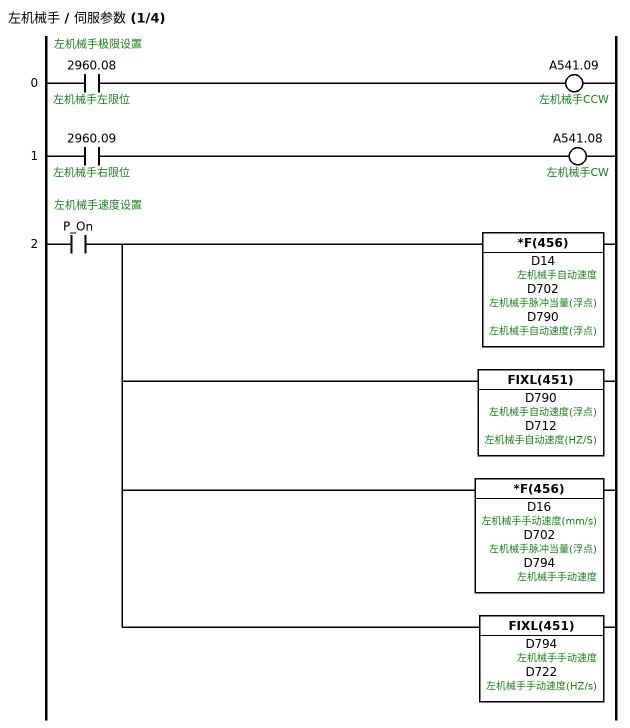
; [picture p137: 左机械手 / 伺服参数, rungs 0-2]
; rung 0: 左机械手极限设置
LD 2960.08  ; 左机械手左限位
OUT A541.09  ; 左机械手CCW
; rung 1
LD 2960.09  ; 左机械手右限位
OUT A541.08  ; 左机械手CW
; rung 2: 左机械手速度设置
LD P_On
*F(456) D14 D702 D790  ; 左机械手自动速度, 左机械手脉冲当量(浮点), 左机械手自动速度(浮点)
FIXL(451) D790 D712  ; 左机械手自动速度(浮点), 左机械手自动速度(HZ/S)
*F(456) D16 D702 D794  ; 左机械手手动速度(mm/s), 左机械手脉冲当量(浮点), 左机械手手动速度
FIXL(451) D794 D722  ; 左机械手手动速度, 左机械手手动速度(HZ/s)

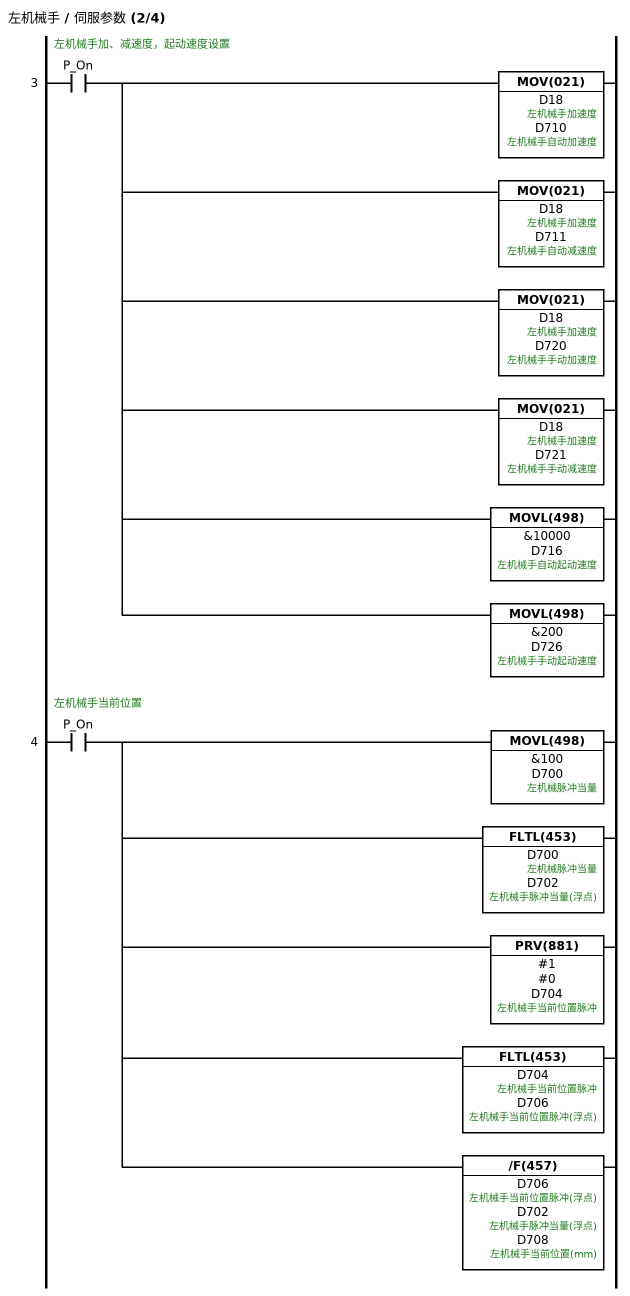
; rung 3: 左机械手加、减速度，起动速度设置
LD P_On
MOV(021) D18 D710  ; 左机械手加速度, 左机械手自动加速度
MOV(021) D18 D711  ; 左机械手加速度, 左机械手自动减速度
MOV(021) D18 D720  ; 左机械手加速度, 左机械手手动加速度
MOV(021) D18 D721  ; 左机械手加速度, 左机械手手动减速度
MOVL(498) &10000 D716  ; 左机械手自动起动速度
MOVL(498) &200 D726  ; 左机械手手动起动速度
; rung 4: 左机械手当前位置
LD P_On
MOVL(498) &100 D700  ; 左机械脉冲当量
FLTL(453) D700 D702  ; 左机械脉冲当量, 左机械手脉冲当量(浮点)
PRV(881) #1 #0 D704  ; 左机械手当前位置脉冲
FLTL(453) D704 D706  ; 左机械手当前位置脉冲, 左机械手当前位置脉冲(浮点)
/F(457) D706 D702 D708  ; 左机械手当前位置脉冲(浮点), 左机械手脉冲当量(浮点), 左机械手当前位置(mm)

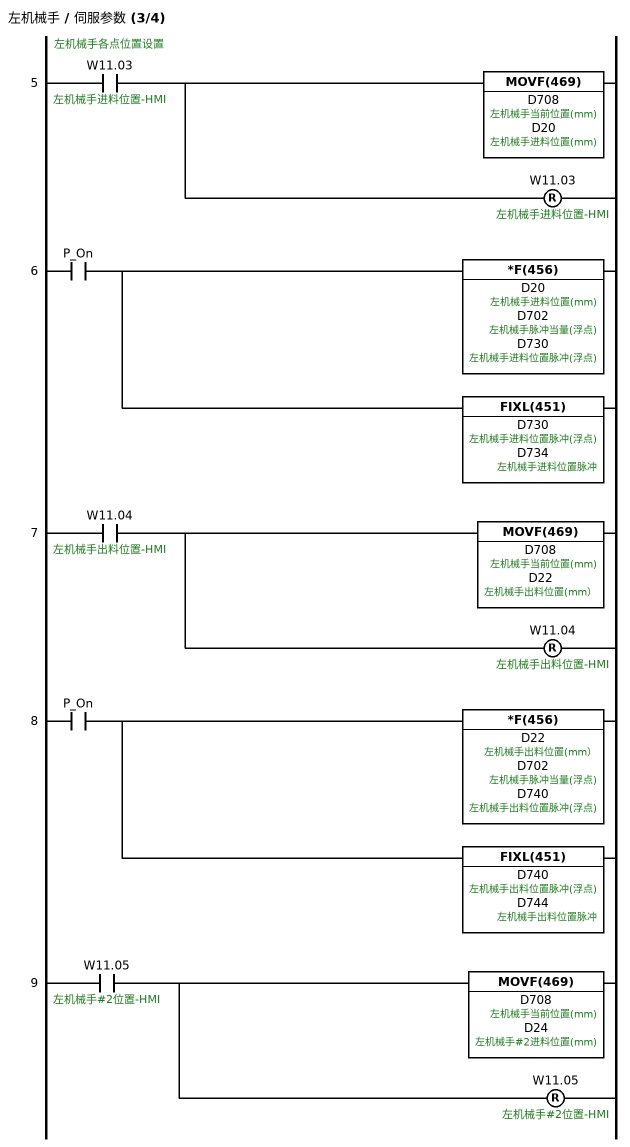
; rung 5: 左机械手各点位置设置
LD W11.03  ; 左机械手进料位置-HMI
MOVF(469) D708 D20  ; 左机械手当前位置(mm), 左机械手进料位置(mm)
RSET W11.03  ; 左机械手进料位置-HMI
; rung 6
LD P_On
*F(456) D20 D702 D730  ; 左机械手进料位置(mm), 左机械手脉冲当量(浮点), 左机械手进料位置脉冲(浮点)
FIXL(451) D730 D734  ; 左机械手进料位置脉冲(浮点), 左机械手进料位置脉冲
; rung 7
LD W11.04  ; 左机械手出料位置-HMI
MOVF(469) D708 D22  ; 左机械手当前位置(mm), 左机械手出料位置(mm）
RSET W11.04  ; 左机械手出料位置-HMI
; rung 8
LD P_On
*F(456) D22 D702 D740  ; 左机械手出料位置(mm）, 左机械手脉冲当量(浮点), 左机械手出料位置脉冲(浮点)
FIXL(451) D740 D744  ; 左机械手出料位置脉冲(浮点), 左机械手出料位置脉冲
; rung 9
LD W11.05  ; 左机械手#2位置-HMI
MOVF(469) D708 D24  ; 左机械手当前位置(mm), 左机械手#2进料位置(mm)
RSET W11.05  ; 左机械手#2位置-HMI

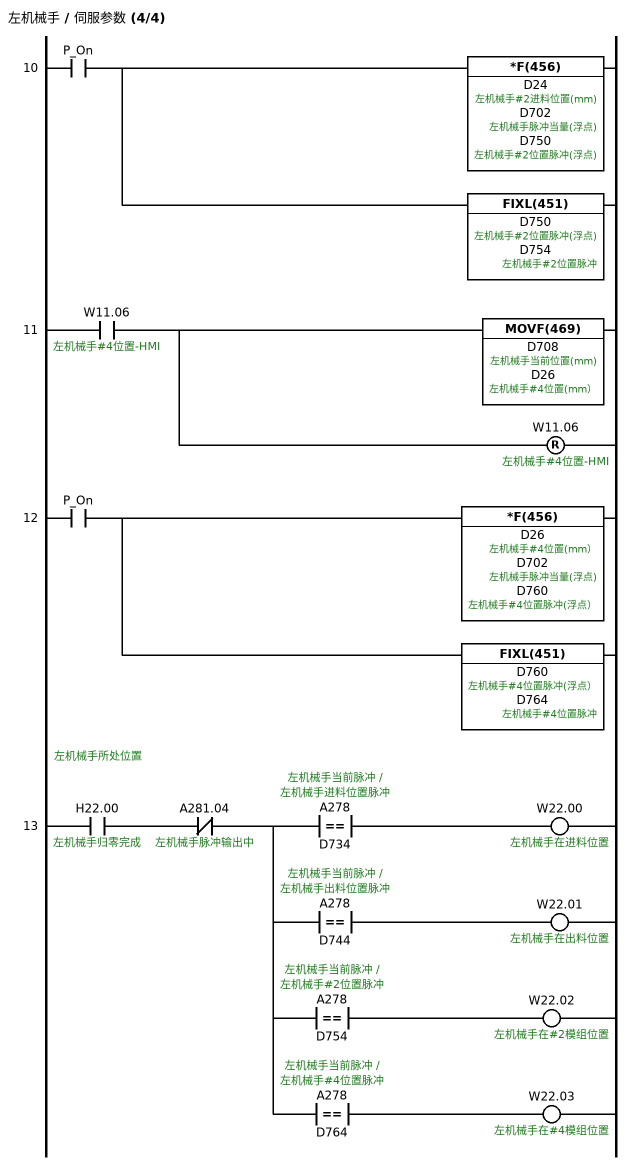
; rung 10
LD P_On
*F(456) D24 D702 D750  ; 左机械手#2进料位置(mm), 左机械手脉冲当量(浮点), 左机械手#2位置脉冲(浮点)
FIXL(451) D750 D754  ; 左机械手#2位置脉冲(浮点), 左机械手#2位置脉冲
; rung 11
LD W11.06  ; 左机械手#4位置-HMI
MOVF(469) D708 D26  ; 左机械手当前位置(mm), 左机械手#4位置(mm）
RSET W11.06  ; 左机械手#4位置-HMI
; rung 12
LD P_On
*F(456) D26 D702 D760  ; 左机械手#4位置(mm）, 左机械手脉冲当量(浮点), 左机械手#4位置脉冲(浮点）
FIXL(451) D760 D764  ; 左机械手#4位置脉冲(浮点）, 左机械手#4位置脉冲
; rung 13: 左机械手所处位置
LD H22.00  ; 左机械手归零完成
ANDNOT A281.04  ; 左机械手脉冲输出中
OUT TR0
AND=SL(303) A278 D734  ; 左机械手当前脉冲, 左机械手进料位置脉冲
OUT W22.00  ; 左机械手在进料位置
LD TR0
AND=SL(303) A278 D744  ; 左机械手当前脉冲, 左机械手出料位置脉冲
OUT W22.01  ; 左机械手在出料位置
LD TR0
AND=SL(303) A278 D754  ; 左机械手当前脉冲, 左机械手#2位置脉冲
OUT W22.02  ; 左机械手在#2模组位置
LD TR0
AND=SL(303) A278 D764  ; 左机械手当前脉冲, 左机械手#4位置脉冲
OUT W22.03  ; 左机械手在#4模组位置

### Section 轴控运动及外部输出

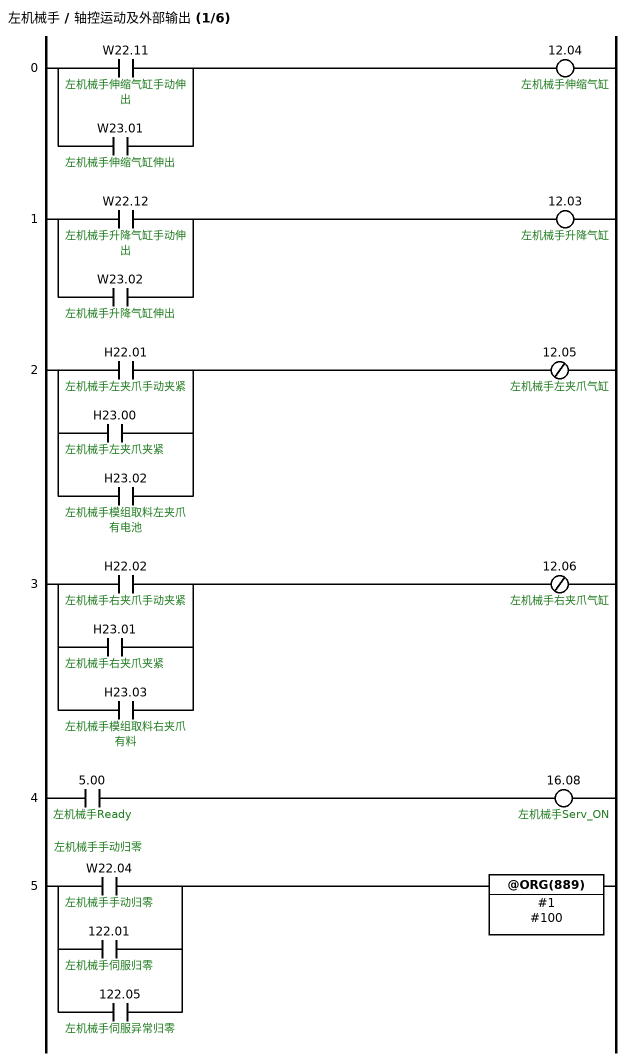
; rung 0
LD W22.11  ; 左机械手伸缩气缸手动伸出
OR W23.01  ; 左机械手伸缩气缸伸出
OUT 12.04  ; 左机械手伸缩气缸
; rung 1
LD W22.12  ; 左机械手升降气缸手动伸出
OR W23.02  ; 左机械手升降气缸伸出
OUT 12.03  ; 左机械手升降气缸
; rung 2
LD H22.01  ; 左机械手左夹爪手动夹紧
OR H23.00  ; 左机械手左夹爪夹紧
OR H23.02  ; 左机械手模组取料左夹爪有电池
OUTNOT 12.05  ; 左机械手左夹爪气缸
; rung 3
LD H22.02  ; 左机械手右夹爪手动夹紧
OR H23.01  ; 左机械手右夹爪夹紧
OR H23.03  ; 左机械手模组取料右夹爪有料
OUTNOT 12.06  ; 左机械手右夹爪气缸
; rung 4
LD 5.00  ; 左机械手Ready
OUT 16.08  ; 左机械手Serv_ON
; rung 5: 左机械手手动归零
LD W22.04  ; 左机械手手动归零
OR 122.01  ; 左机械手伺服归零
OR 122.05  ; 左机械手伺服异常归零
@ORG(889) #1 #100

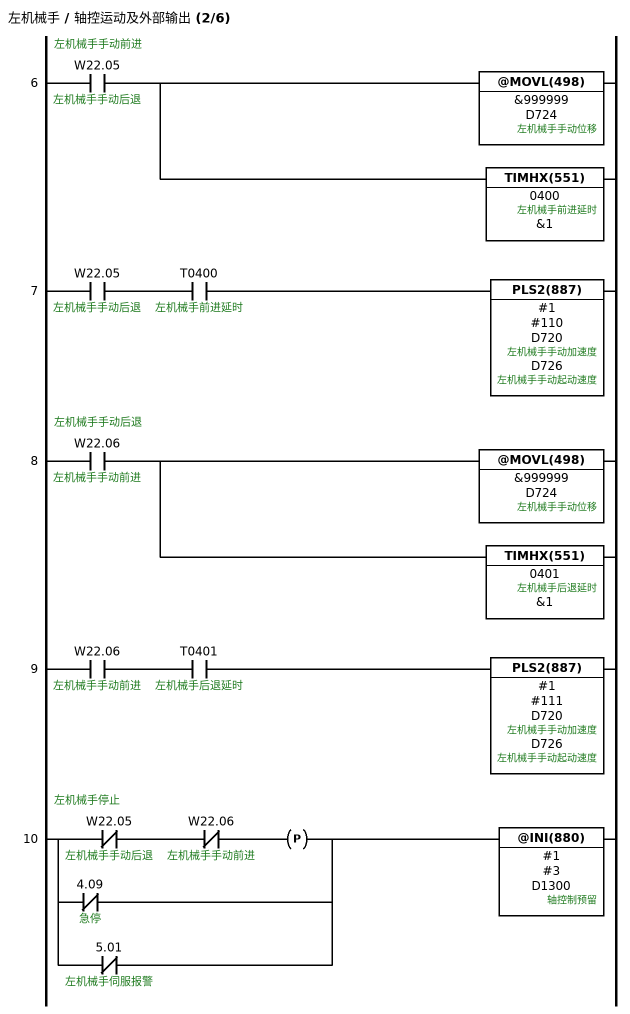
; rung 6: 左机械手手动前进
LD W22.05  ; 左机械手手动后退
@MOVL(498) &999999 D724  ; 左机械手手动位移
TIMHX(551) 0400 &1  ; 左机械手前进延时
; rung 7
LD W22.05  ; 左机械手手动后退
AND T0400  ; 左机械手前进延时
PLS2(887) #1 #110 D720 D726  ; 左机械手手动加速度, 左机械手手动起动速度
; rung 8: 左机械手手动后退
LD W22.06  ; 左机械手手动前进
@MOVL(498) &999999 D724  ; 左机械手手动位移
TIMHX(551) 0401 &1  ; 左机械手后退延时
; rung 9
LD W22.06  ; 左机械手手动前进
AND T0401  ; 左机械手后退延时
PLS2(887) #1 #111 D720 D726  ; 左机械手手动加速度, 左机械手手动起动速度
; rung 10: 左机械手停止
LDNOT W22.05  ; 左机械手手动后退
ANDNOT W22.06  ; 左机械手手动前进
UP(521)
ORNOT 4.09  ; 急停
ORNOT 5.01  ; 左机械手伺服报警
@INI(880) #1 #3 D1300  ; 轴控制预留

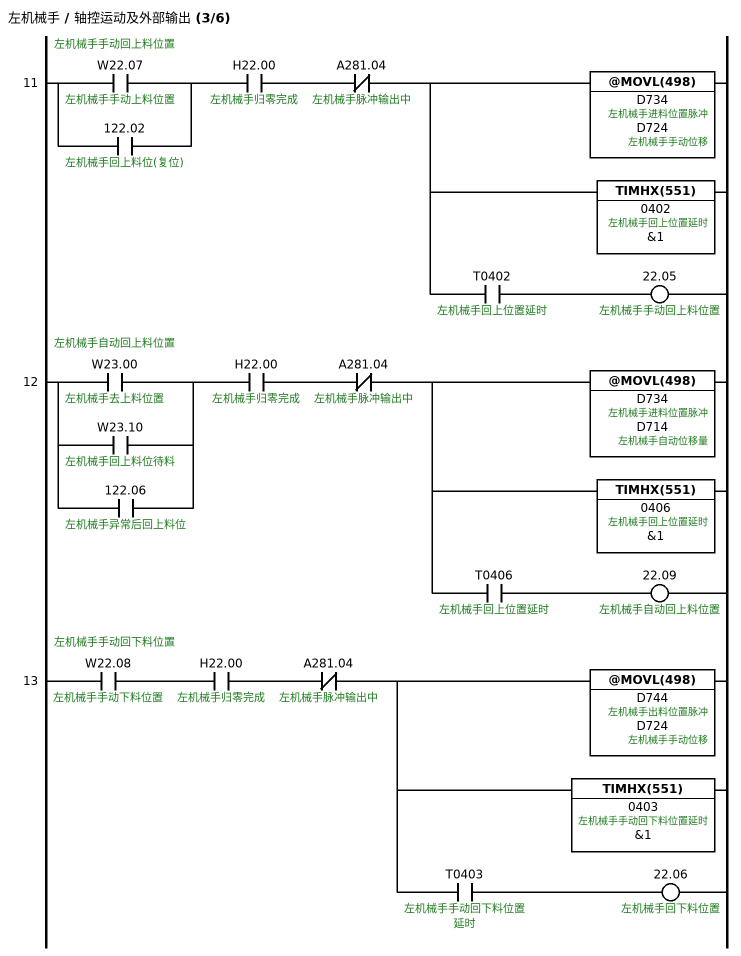
; rung 11: 左机械手手动回上料位置
LD W22.07  ; 左机械手手动上料位置
OR 122.02  ; 左机械手回上料位(复位)
AND H22.00  ; 左机械手归零完成
ANDNOT A281.04  ; 左机械手脉冲输出中
@MOVL(498) D734 D724  ; 左机械手进料位置脉冲, 左机械手手动位移
TIMHX(551) 0402 &1  ; 左机械手回上位置延时
AND T0402  ; 左机械手回上位置延时
OUT 22.05  ; 左机械手手动回上料位置
; rung 12: 左机械手自动回上料位置
LD W23.00  ; 左机械手去上料位置
OR W23.10  ; 左机械手回上料位待料
OR 122.06  ; 左机械手异常后回上料位
AND H22.00  ; 左机械手归零完成
ANDNOT A281.04  ; 左机械手脉冲输出中
@MOVL(498) D734 D714  ; 左机械手进料位置脉冲, 左机械手自动位移量
TIMHX(551) 0406 &1  ; 左机械手回上位置延时
AND T0406  ; 左机械手回上位置延时
OUT 22.09  ; 左机械手自动回上料位置
; rung 13: 左机械手手动回下料位置
LD W22.08  ; 左机械手手动下料位置
AND H22.00  ; 左机械手归零完成
ANDNOT A281.04  ; 左机械手脉冲输出中
@MOVL(498) D744 D724  ; 左机械手出料位置脉冲, 左机械手手动位移
TIMHX(551) 0403 &1  ; 左机械手手动回下料位置延时
AND T0403  ; 左机械手手动回下料位置延时
OUT 22.06  ; 左机械手回下料位置

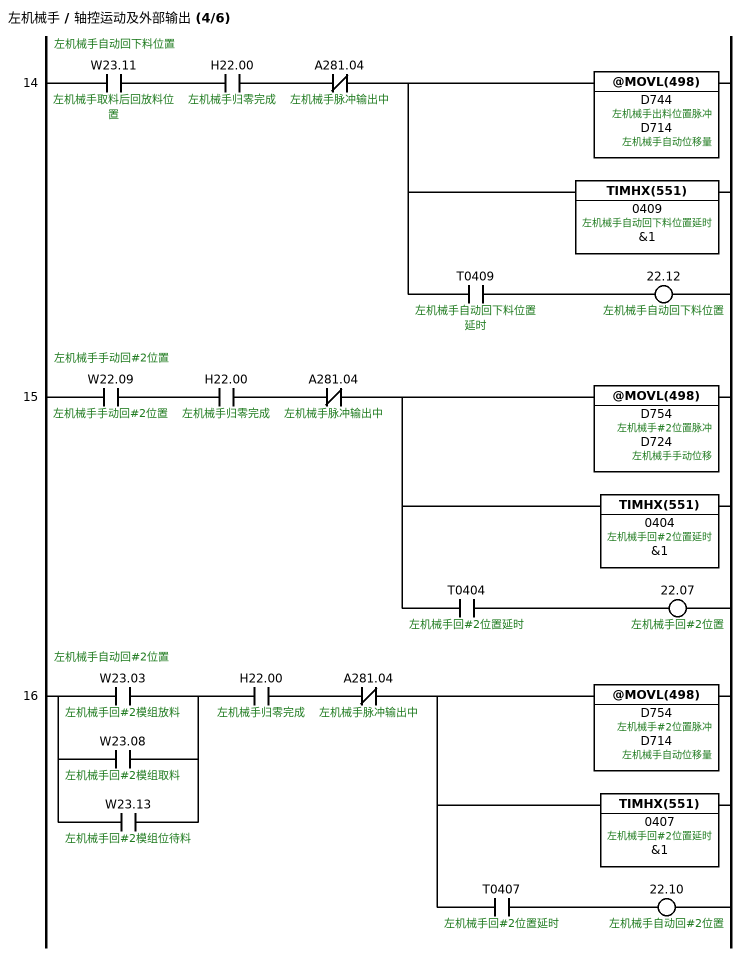
; rung 14: 左机械手自动回下料位置
LD W23.11  ; 左机械手取料后回放料位置
AND H22.00  ; 左机械手归零完成
ANDNOT A281.04  ; 左机械手脉冲输出中
@MOVL(498) D744 D714  ; 左机械手出料位置脉冲, 左机械手自动位移量
TIMHX(551) 0409 &1  ; 左机械手自动回下料位置延时
AND T0409  ; 左机械手自动回下料位置延时
OUT 22.12  ; 左机械手自动回下料位置
; rung 15: 左机械手手动回#2位置
LD W22.09  ; 左机械手手动回#2位置
AND H22.00  ; 左机械手归零完成
ANDNOT A281.04  ; 左机械手脉冲输出中
@MOVL(498) D754 D724  ; 左机械手#2位置脉冲, 左机械手手动位移
TIMHX(551) 0404 &1  ; 左机械手回#2位置延时
AND T0404  ; 左机械手回#2位置延时
OUT 22.07  ; 左机械手回#2位置
; rung 16: 左机械手自动回#2位置
LD W23.03  ; 左机械手回#2模组放料
OR W23.08  ; 左机械手回#2模组取料
OR W23.13  ; 左机械手回#2模组位待料
AND H22.00  ; 左机械手归零完成
ANDNOT A281.04  ; 左机械手脉冲输出中
@MOVL(498) D754 D714  ; 左机械手#2位置脉冲, 左机械手自动位移量
TIMHX(551) 0407 &1  ; 左机械手回#2位置延时
AND T0407  ; 左机械手回#2位置延时
OUT 22.10  ; 左机械手自动回#2位置

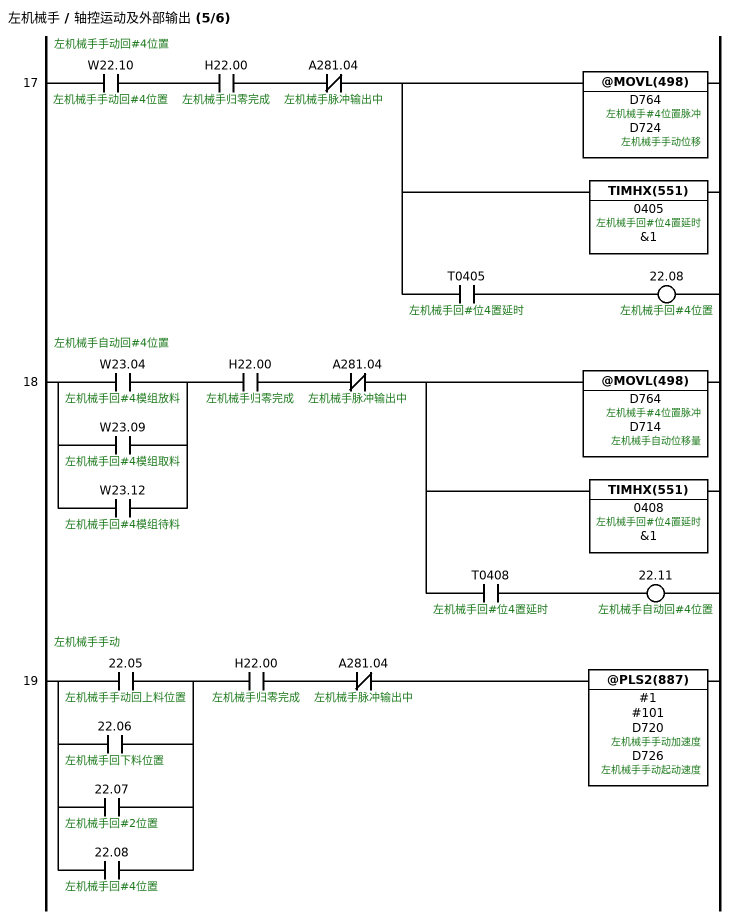
; rung 17: 左机械手手动回#4位置
LD W22.10  ; 左机械手手动回#4位置
AND H22.00  ; 左机械手归零完成
ANDNOT A281.04  ; 左机械手脉冲输出中
@MOVL(498) D764 D724  ; 左机械手#4位置脉冲, 左机械手手动位移
TIMHX(551) 0405 &1  ; 左机械手回#位4置延时
AND T0405  ; 左机械手回#位4置延时
OUT 22.08  ; 左机械手回#4位置
; rung 18: 左机械手自动回#4位置
LD W23.04  ; 左机械手回#4模组放料
OR W23.09  ; 左机械手回#4模组取料
OR W23.12  ; 左机械手回#4模组待料
AND H22.00  ; 左机械手归零完成
ANDNOT A281.04  ; 左机械手脉冲输出中
@MOVL(498) D764 D714  ; 左机械手#4位置脉冲, 左机械手自动位移量
TIMHX(551) 0408 &1  ; 左机械手回#位4置延时
AND T0408  ; 左机械手回#位4置延时
OUT 22.11  ; 左机械手自动回#4位置
; rung 19: 左机械手手动
LD 22.05  ; 左机械手手动回上料位置
OR 22.06  ; 左机械手回下料位置
OR 22.07  ; 左机械手回#2位置
OR 22.08  ; 左机械手回#4位置
AND H22.00  ; 左机械手归零完成
ANDNOT A281.04  ; 左机械手脉冲输出中
@PLS2(887) #1 #101 D720 D726  ; 左机械手手动加速度, 左机械手手动起动速度

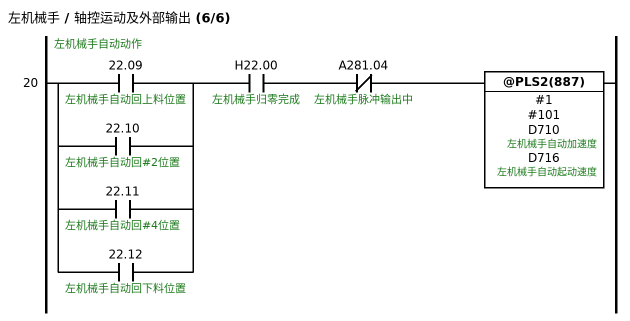
; rung 20: 左机械手自动动作
LD 22.09  ; 左机械手自动回上料位置
OR 22.10  ; 左机械手自动回#2位置
OR 22.11  ; 左机械手自动回#4位置
OR 22.12  ; 左机械手自动回下料位置
AND H22.00  ; 左机械手归零完成
ANDNOT A281.04  ; 左机械手脉冲输出中
@PLS2(887) #1 #101 D710 D716  ; 左机械手自动加速度, 左机械手自动起动速度

### Section 自动报警

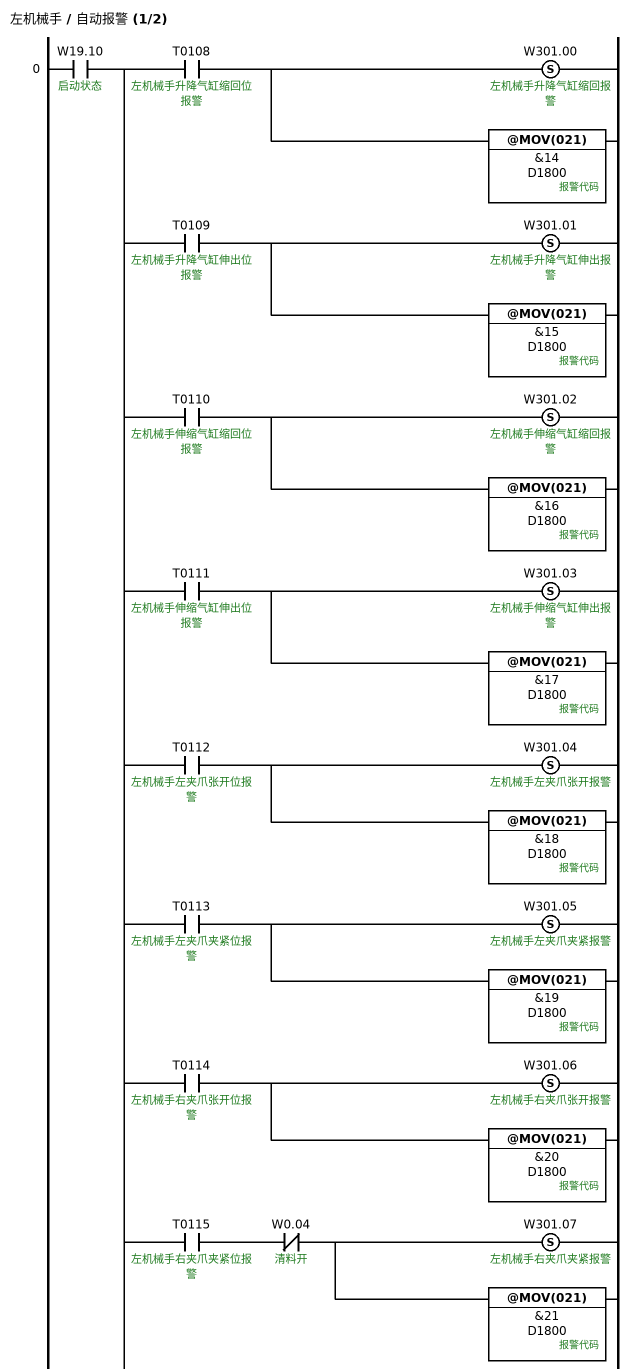

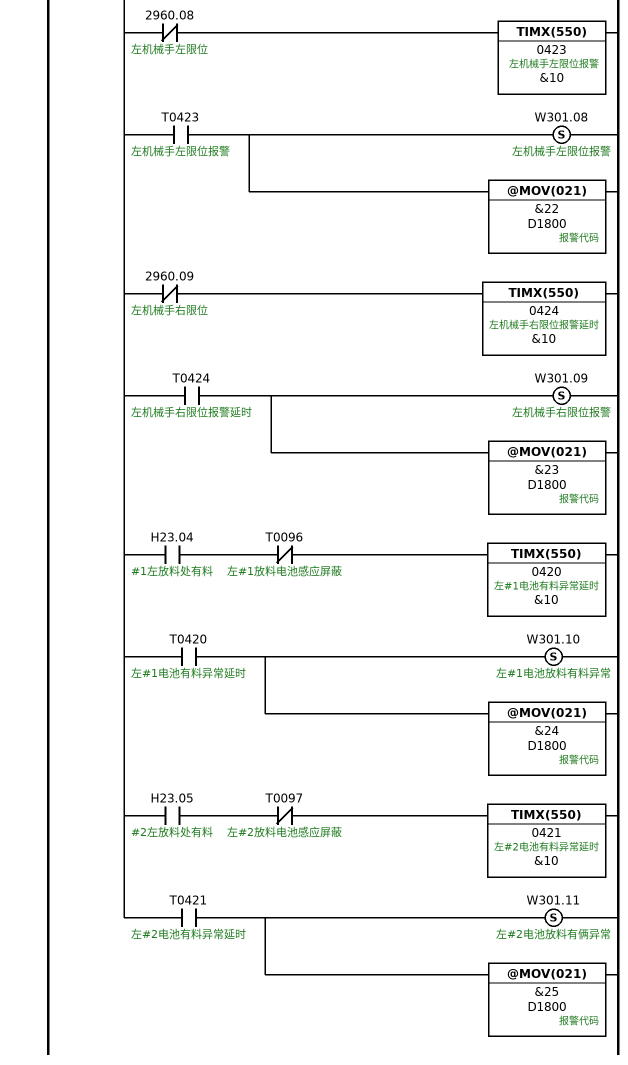
; rung 0
LD W19.10  ; 启动状态
OUT TR0
AND T0108  ; 左机械手升降气缸缩回位报警
SET W301.00  ; 左机械手升降气缸缩回报警
@MOV(021) &14 D1800  ; 报警代码
LD TR0
AND T0109  ; 左机械手升降气缸伸出位报警
SET W301.01  ; 左机械手升降气缸伸出报警
@MOV(021) &15 D1800  ; 报警代码
LD TR0
AND T0110  ; 左机械手伸缩气缸缩回位报警
SET W301.02  ; 左机械手伸缩气缸缩回报警
@MOV(021) &16 D1800  ; 报警代码
LD TR0
AND T0111  ; 左机械手伸缩气缸伸出位报警
SET W301.03  ; 左机械手伸缩气缸伸出报警
@MOV(021) &17 D1800  ; 报警代码
LD TR0
AND T0112  ; 左机械手左夹爪张开位报警
SET W301.04  ; 左机械手左夹爪张开报警
@MOV(021) &18 D1800  ; 报警代码
LD TR0
AND T0113  ; 左机械手左夹爪夹紧位报警
SET W301.05  ; 左机械手左夹爪夹紧报警
@MOV(021) &19 D1800  ; 报警代码
LD TR0
AND T0114  ; 左机械手右夹爪张开位报警
SET W301.06  ; 左机械手右夹爪张开报警
@MOV(021) &20 D1800  ; 报警代码
LD TR0
AND T0115  ; 左机械手右夹爪夹紧位报警
ANDNOT W0.04  ; 清料开
SET W301.07  ; 左机械手右夹爪夹紧报警
@MOV(021) &21 D1800  ; 报警代码
LD TR0
ANDNOT 2960.08  ; 左机械手左限位
TIMX(550) 0423 &10  ; 左机械手左限位报警
LD TR0
AND T0423  ; 左机械手左限位报警
SET W301.08  ; 左机械手左限位报警
@MOV(021) &22 D1800  ; 报警代码
LD TR0
ANDNOT 2960.09  ; 左机械手右限位
TIMX(550) 0424 &10  ; 左机械手右限位报警延时
LD TR0
AND T0424  ; 左机械手右限位报警延时
SET W301.09  ; 左机械手右限位报警
@MOV(021) &23 D1800  ; 报警代码
LD TR0
AND H23.04  ; #1左放料处有料
ANDNOT T0096  ; 左#1放料电池感应屏蔽
TIMX(550) 0420 &10  ; 左#1电池有料异常延时
LD TR0
AND T0420  ; 左#1电池有料异常延时
SET W301.10  ; 左#1电池放料有料异常
@MOV(021) &24 D1800  ; 报警代码
LD TR0
AND H23.05  ; #2左放料处有料
ANDNOT T0097  ; 左#2放料电池感应屏蔽
TIMX(550) 0421 &10  ; 左#2电池有料异常延时
LD TR0
AND T0421  ; 左#2电池有料异常延时
SET W301.11  ; 左#2电池放料有俩异常
@MOV(021) &25 D1800  ; 报警代码

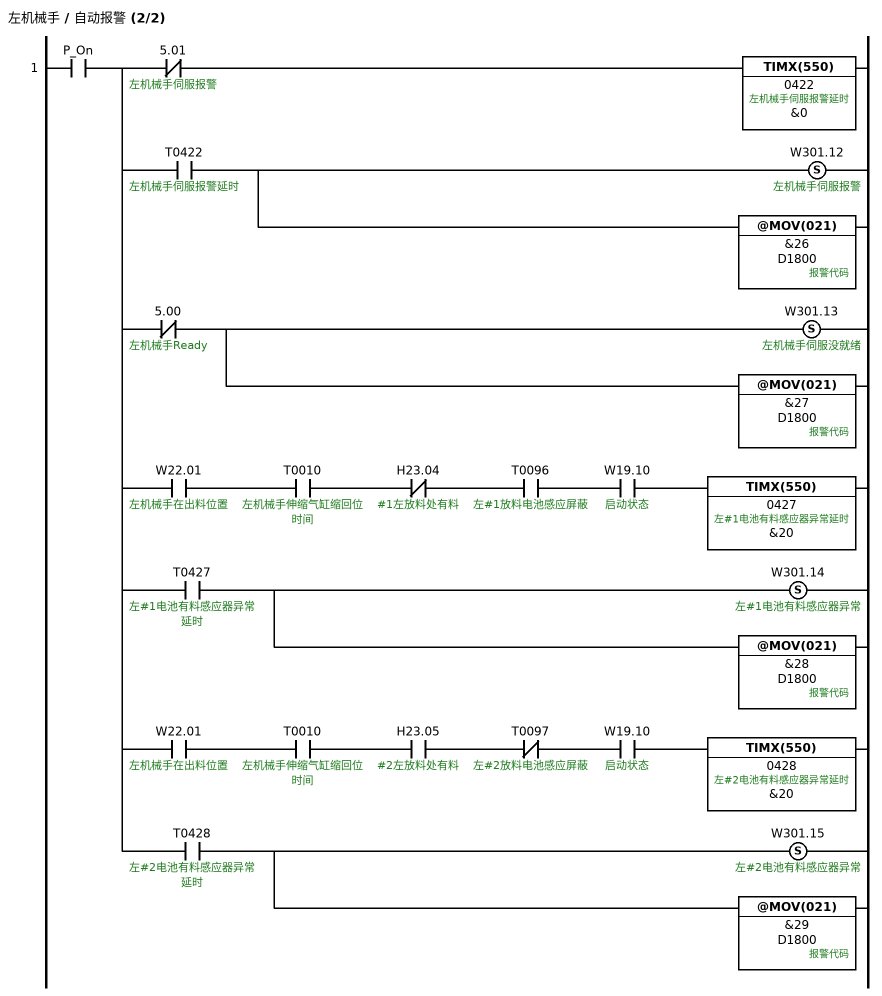
; rung 1
LD P_On
OUT TR0
ANDNOT 5.01  ; 左机械手伺服报警
TIMX(550) 0422 &0  ; 左机械手伺服报警延时
LD TR0
AND T0422  ; 左机械手伺服报警延时
SET W301.12  ; 左机械手伺服报警
@MOV(021) &26 D1800  ; 报警代码
LD TR0
ANDNOT 5.00  ; 左机械手Ready
SET W301.13  ; 左机械手伺服没就绪
@MOV(021) &27 D1800  ; 报警代码
LD TR0
AND W22.01  ; 左机械手在出料位置
AND T0010  ; 左机械手伸缩气缸缩回位时间
ANDNOT H23.04  ; #1左放料处有料
AND T0096  ; 左#1放料电池感应屏蔽
AND W19.10  ; 启动状态
TIMX(550) 0427 &20  ; 左#1电池有料感应器异常延时
LD TR0
AND T0427  ; 左#1电池有料感应器异常延时
SET W301.14  ; 左#1电池有料感应器异常
@MOV(021) &28 D1800  ; 报警代码
LD TR0
AND W22.01  ; 左机械手在出料位置
AND T0010  ; 左机械手伸缩气缸缩回位时间
AND H23.05  ; #2左放料处有料
ANDNOT T0097  ; 左#2放料电池感应屏蔽
AND W19.10  ; 启动状态
TIMX(550) 0428 &20  ; 左#2电池有料感应器异常延时
LD TR0
AND T0428  ; 左#2电池有料感应器异常延时
SET W301.15  ; 左#2电池有料感应器异常
@MOV(021) &29 D1800  ; 报警代码

### Section 左机械手复位

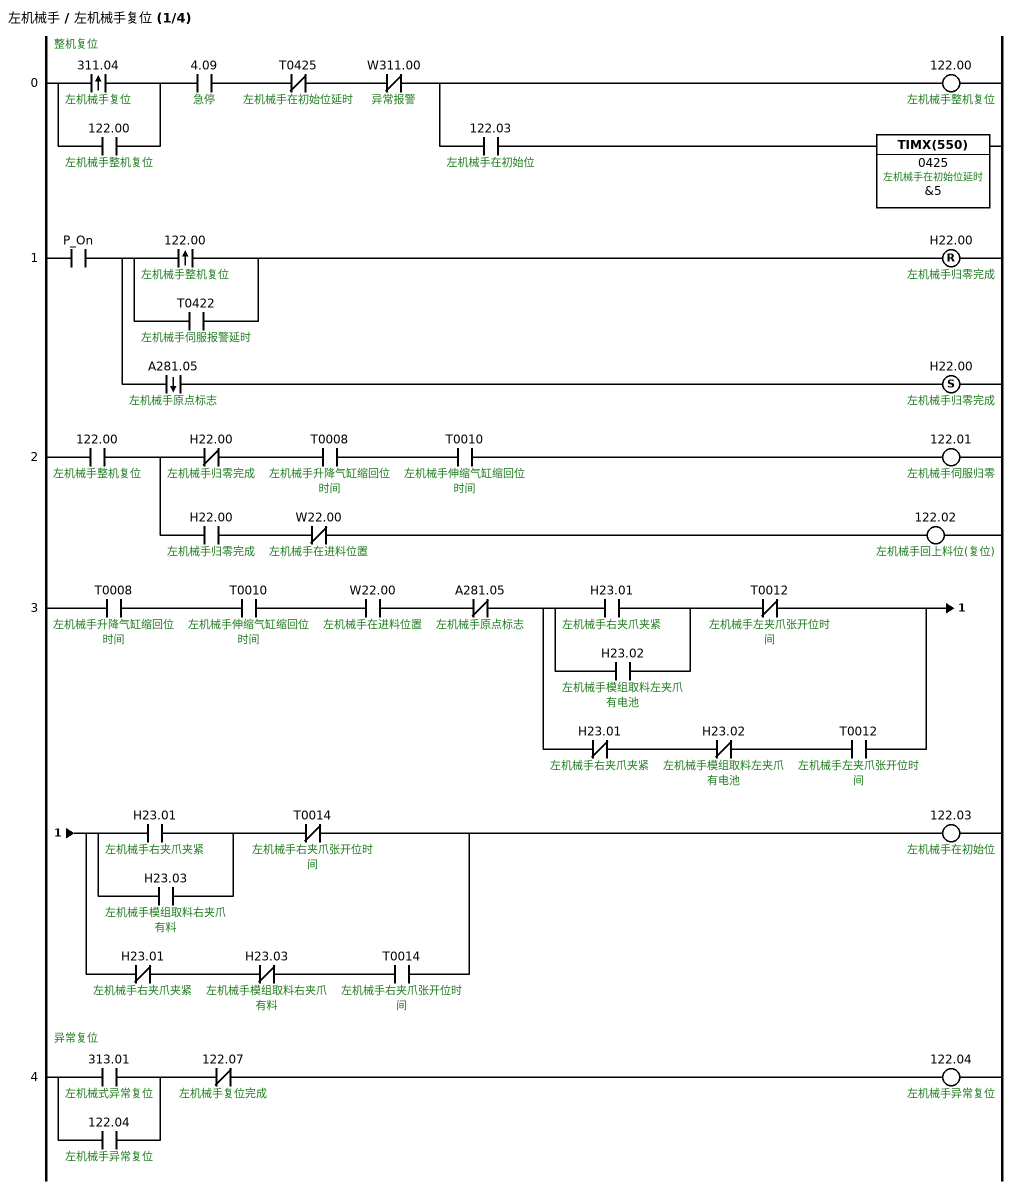
; rung 0: 整机复位
@LD 311.04  ; 左机械手复位
OR 122.00  ; 左机械手整机复位
AND 4.09  ; 急停
ANDNOT T0425  ; 左机械手在初始位延时
ANDNOT W311.00  ; 异常报警
OUT 122.00  ; 左机械手整机复位
AND 122.03  ; 左机械手在初始位
TIMX(550) 0425 &5  ; 左机械手在初始位延时
; rung 1
LD P_On
OUT TR0
@LD 122.00  ; 左机械手整机复位
OR T0422  ; 左机械手伺服报警延时
ANDLD
RSET H22.00  ; 左机械手归零完成
LD TR0
%AND A281.05  ; 左机械手原点标志
SET H22.00  ; 左机械手归零完成
; rung 2
LD 122.00  ; 左机械手整机复位
OUT TR0
ANDNOT H22.00  ; 左机械手归零完成
AND T0008  ; 左机械手升降气缸缩回位时间
AND T0010  ; 左机械手伸缩气缸缩回位时间
OUT 122.01  ; 左机械手伺服归零
LD TR0
AND H22.00  ; 左机械手归零完成
ANDNOT W22.00  ; 左机械手在进料位置
OUT 122.02  ; 左机械手回上料位(复位)
; rung 3
LD T0008  ; 左机械手升降气缸缩回位时间
AND T0010  ; 左机械手伸缩气缸缩回位时间
AND W22.00  ; 左机械手在进料位置
ANDNOT A281.05  ; 左机械手原点标志
LD H23.01  ; 左机械手右夹爪夹紧
OR H23.02  ; 左机械手模组取料左夹爪有电池
ANDNOT T0012  ; 左机械手左夹爪张开位时间
LDNOT H23.01  ; 左机械手右夹爪夹紧
ANDNOT H23.02  ; 左机械手模组取料左夹爪有电池
AND T0012  ; 左机械手左夹爪张开位时间
ORLD
ANDLD
LD H23.01  ; 左机械手右夹爪夹紧
OR H23.03  ; 左机械手模组取料右夹爪有料
ANDNOT T0014  ; 左机械手右夹爪张开位时间
LDNOT H23.01  ; 左机械手右夹爪夹紧
ANDNOT H23.03  ; 左机械手模组取料右夹爪有料
AND T0014  ; 左机械手右夹爪张开位时间
ORLD
ANDLD
OUT 122.03  ; 左机械手在初始位
; rung 4: 异常复位
LD 313.01  ; 左机械式异常复位
OR 122.04  ; 左机械手异常复位
ANDNOT 122.07  ; 左机械手复位完成
OUT 122.04  ; 左机械手异常复位

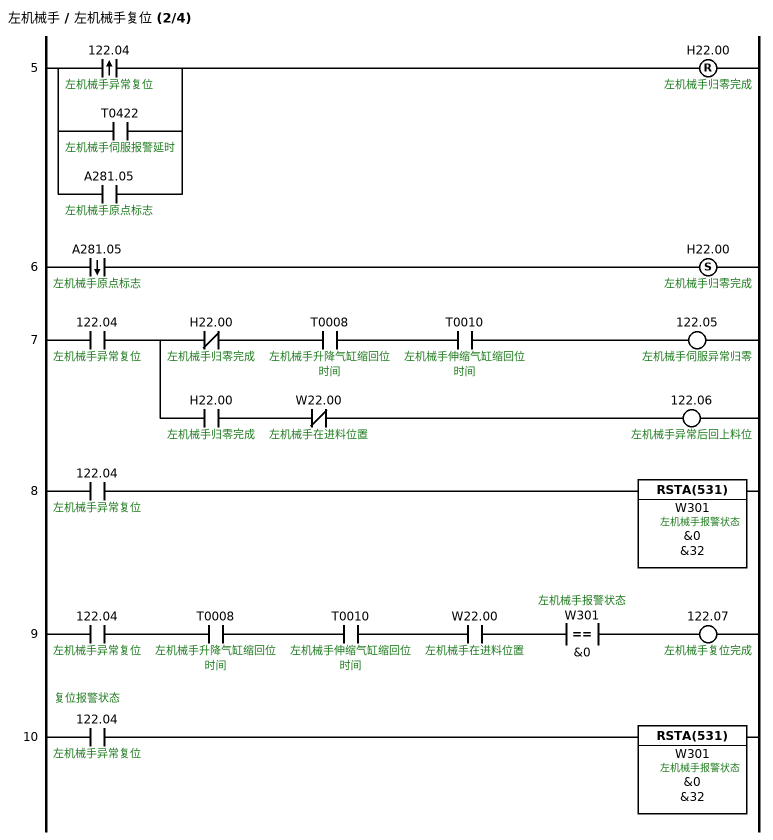
; rung 5
@LD 122.04  ; 左机械手异常复位
OR T0422  ; 左机械手伺服报警延时
OR A281.05  ; 左机械手原点标志
RSET H22.00  ; 左机械手归零完成
; rung 6
%LD A281.05  ; 左机械手原点标志
SET H22.00  ; 左机械手归零完成
; rung 7
LD 122.04  ; 左机械手异常复位
OUT TR0
ANDNOT H22.00  ; 左机械手归零完成
AND T0008  ; 左机械手升降气缸缩回位时间
AND T0010  ; 左机械手伸缩气缸缩回位时间
OUT 122.05  ; 左机械手伺服异常归零
LD TR0
AND H22.00  ; 左机械手归零完成
ANDNOT W22.00  ; 左机械手在进料位置
OUT 122.06  ; 左机械手异常后回上料位
; rung 8
LD 122.04  ; 左机械手异常复位
RSTA(531) W301 &0 &32  ; 左机械手报警状态
; rung 9
LD 122.04  ; 左机械手异常复位
AND T0008  ; 左机械手升降气缸缩回位时间
AND T0010  ; 左机械手伸缩气缸缩回位时间
AND W22.00  ; 左机械手在进料位置
AND=L(301) W301 &0  ; 左机械手报警状态
OUT 122.07  ; 左机械手复位完成
; rung 10: 复位报警状态
LD 122.04  ; 左机械手异常复位
RSTA(531) W301 &0 &32  ; 左机械手报警状态

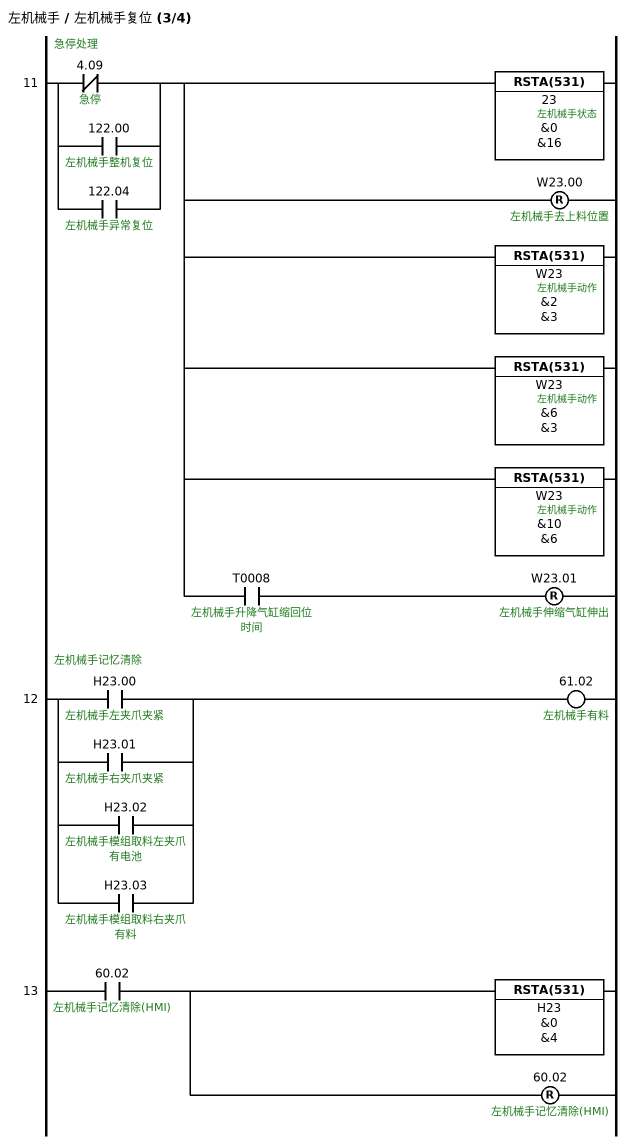
; rung 11: 急停处理
LDNOT 4.09  ; 急停
OR 122.00  ; 左机械手整机复位
OR 122.04  ; 左机械手异常复位
RSTA(531) 23 &0 &16  ; 左机械手状态
RSET W23.00  ; 左机械手去上料位置
RSTA(531) W23 &2 &3  ; 左机械手动作
RSTA(531) W23 &6 &3  ; 左机械手动作
RSTA(531) W23 &10 &6  ; 左机械手动作
AND T0008  ; 左机械手升降气缸缩回位时间
RSET W23.01  ; 左机械手伸缩气缸伸出
; rung 12: 左机械手记忆清除
LD H23.00  ; 左机械手左夹爪夹紧
OR H23.01  ; 左机械手右夹爪夹紧
OR H23.02  ; 左机械手模组取料左夹爪有电池
OR H23.03  ; 左机械手模组取料右夹爪有料
OUT 61.02  ; 左机械手有料
; rung 13
LD 60.02  ; 左机械手记忆清除(HMI)
RSTA(531) H23 &0 &4
RSET 60.02  ; 左机械手记忆清除(HMI)

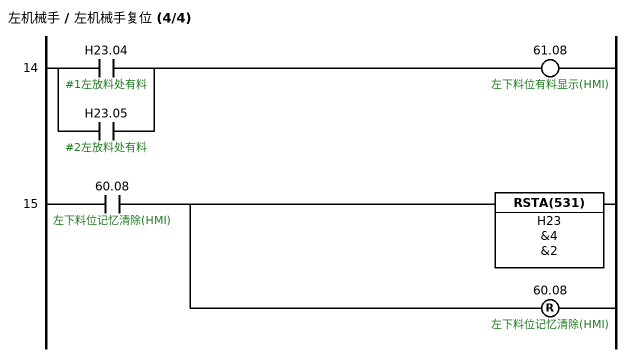
; rung 14
LD H23.04  ; #1左放料处有料
OR H23.05  ; #2左放料处有料
OUT 61.08  ; 左下料位有料显示(HMI)
; rung 15
LD 60.08  ; 左下料位记忆清除(HMI)
RSTA(531) H23 &4 &2
RSET 60.08  ; 左下料位记忆清除(HMI)

### Section END
; rung 0
END(001)

## Program 右机械手 (cyclic task 5)

### Section 右机械手手动

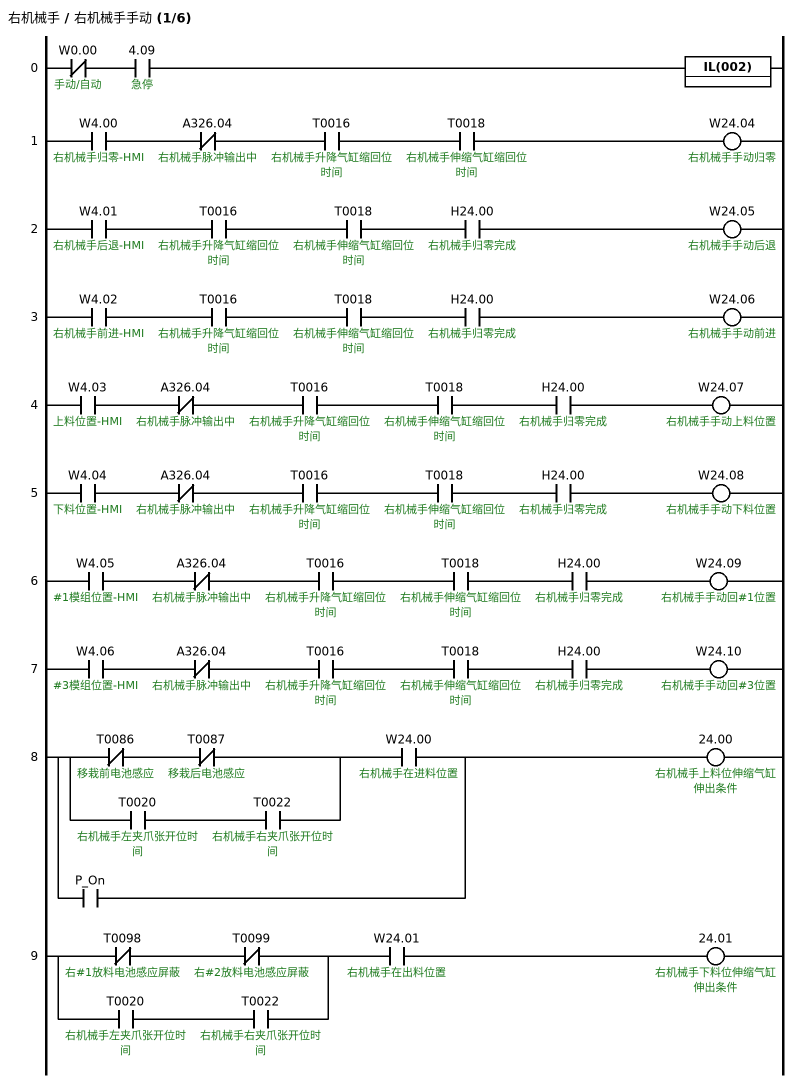
; rung 0
LDNOT W0.00  ; 手动/自动
AND 4.09  ; 急停
IL(002)
; rung 1
LD W4.00  ; 右机械手归零-HMI
ANDNOT A326.04  ; 右机械手脉冲输出中
AND T0016  ; 右机械手升降气缸缩回位时间
AND T0018  ; 右机械手伸缩气缸缩回位时间
OUT W24.04  ; 右机械手手动归零
; rung 2
LD W4.01  ; 右机械手后退-HMI
AND T0016  ; 右机械手升降气缸缩回位时间
AND T0018  ; 右机械手伸缩气缸缩回位时间
AND H24.00  ; 右机械手归零完成
OUT W24.05  ; 右机械手手动后退
; rung 3
LD W4.02  ; 右机械手前进-HMI
AND T0016  ; 右机械手升降气缸缩回位时间
AND T0018  ; 右机械手伸缩气缸缩回位时间
AND H24.00  ; 右机械手归零完成
OUT W24.06  ; 右机械手手动前进
; rung 4
LD W4.03  ; 上料位置-HMI
ANDNOT A326.04  ; 右机械手脉冲输出中
AND T0016  ; 右机械手升降气缸缩回位时间
AND T0018  ; 右机械手伸缩气缸缩回位时间
AND H24.00  ; 右机械手归零完成
OUT W24.07  ; 右机械手手动上料位置
; rung 5
LD W4.04  ; 下料位置-HMI
ANDNOT A326.04  ; 右机械手脉冲输出中
AND T0016  ; 右机械手升降气缸缩回位时间
AND T0018  ; 右机械手伸缩气缸缩回位时间
AND H24.00  ; 右机械手归零完成
OUT W24.08  ; 右机械手手动下料位置
; rung 6
LD W4.05  ; #1模组位置-HMI
ANDNOT A326.04  ; 右机械手脉冲输出中
AND T0016  ; 右机械手升降气缸缩回位时间
AND T0018  ; 右机械手伸缩气缸缩回位时间
AND H24.00  ; 右机械手归零完成
OUT W24.09  ; 右机械手手动回#1位置
; rung 7
LD W4.06  ; #3模组位置-HMI
ANDNOT A326.04  ; 右机械手脉冲输出中
AND T0016  ; 右机械手升降气缸缩回位时间
AND T0018  ; 右机械手伸缩气缸缩回位时间
AND H24.00  ; 右机械手归零完成
OUT W24.10  ; 右机械手手动回#3位置
; rung 8
LDNOT T0086  ; 移栽前电池感应
ANDNOT T0087  ; 移栽后电池感应
LD T0020  ; 右机械手左夹爪张开位时间
AND T0022  ; 右机械手右夹爪张开位时间
ORLD
AND W24.00  ; 右机械手在进料位置
OR P_On
OUT 24.00  ; 右机械手上料位伸缩气缸伸出条件
; rung 9
LDNOT T0098  ; 右#1放料电池感应屏蔽
ANDNOT T0099  ; 右#2放料电池感应屏蔽
LD T0020  ; 右机械手左夹爪张开位时间
AND T0022  ; 右机械手右夹爪张开位时间
ORLD
AND W24.01  ; 右机械手在出料位置
OUT 24.01  ; 右机械手下料位伸缩气缸伸出条件

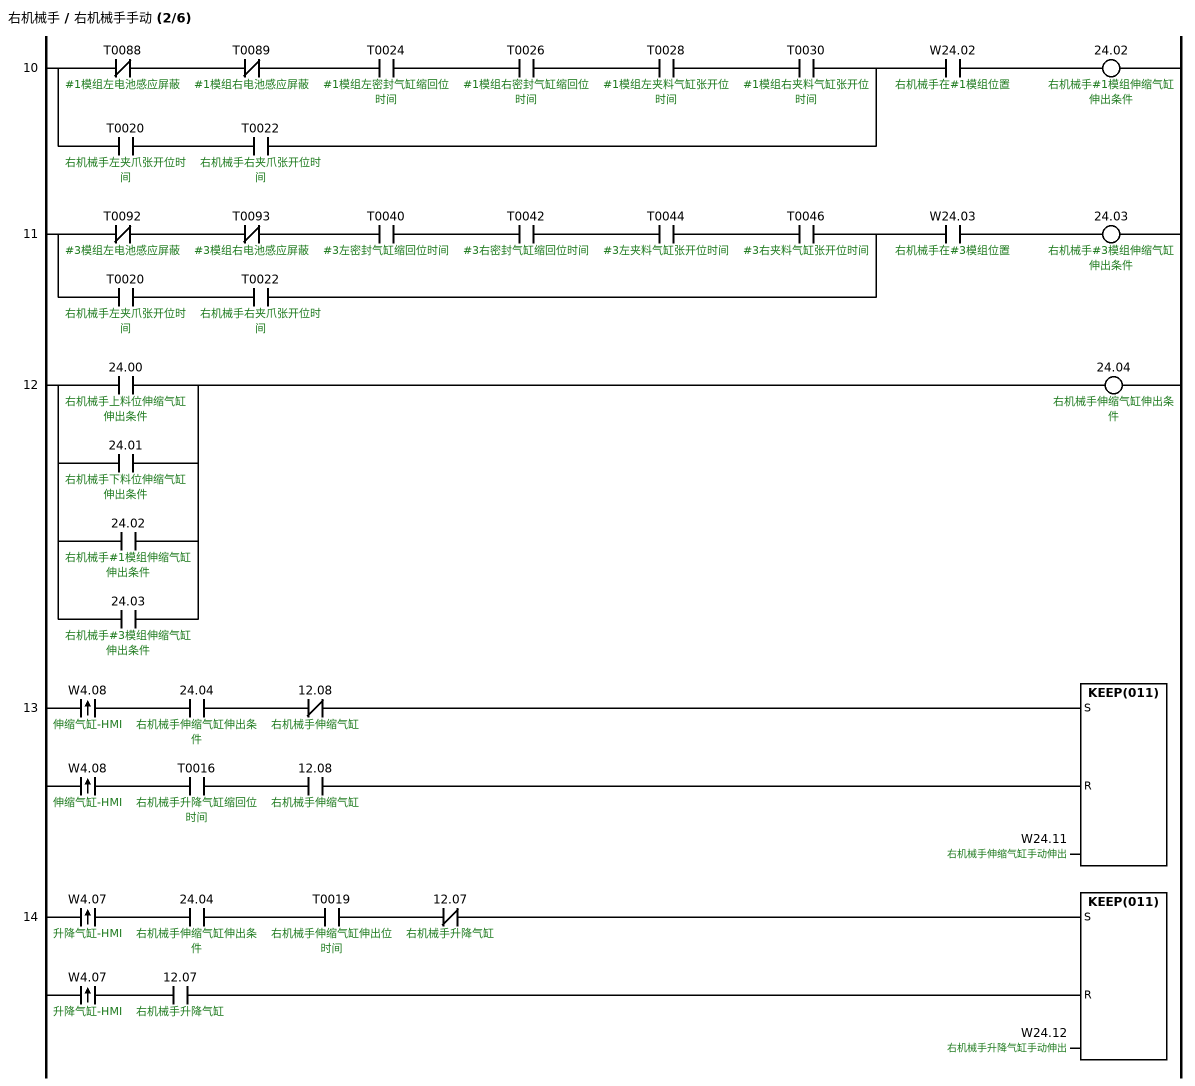
; rung 10
LDNOT T0088  ; #1模组左电池感应屏蔽
ANDNOT T0089  ; #1模组右电池感应屏蔽
AND T0024  ; #1模组左密封气缸缩回位时间
AND T0026  ; #1模组右密封气缸缩回位时间
AND T0028  ; #1模组左夹料气缸张开位时间
AND T0030  ; #1模组右夹料气缸张开位时间
LD T0020  ; 右机械手左夹爪张开位时间
AND T0022  ; 右机械手右夹爪张开位时间
ORLD
AND W24.02  ; 右机械手在#1模组位置
OUT 24.02  ; 右机械手#1模组伸缩气缸伸出条件
; rung 11
LDNOT T0092  ; #3模组左电池感应屏蔽
ANDNOT T0093  ; #3模组右电池感应屏蔽
AND T0040  ; #3左密封气缸缩回位时间
AND T0042  ; #3右密封气缸缩回位时间
AND T0044  ; #3左夹料气缸张开位时间
AND T0046  ; #3右夹料气缸张开位时间
LD T0020  ; 右机械手左夹爪张开位时间
AND T0022  ; 右机械手右夹爪张开位时间
ORLD
AND W24.03  ; 右机械手在#3模组位置
OUT 24.03  ; 右机械手#3模组伸缩气缸伸出条件
; rung 12
LD 24.00  ; 右机械手上料位伸缩气缸伸出条件
OR 24.01  ; 右机械手下料位伸缩气缸伸出条件
OR 24.02  ; 右机械手#1模组伸缩气缸伸出条件
OR 24.03  ; 右机械手#3模组伸缩气缸伸出条件
OUT 24.04  ; 右机械手伸缩气缸伸出条件
; rung 13
@LD W4.08  ; 伸缩气缸-HMI
AND 24.04  ; 右机械手伸缩气缸伸出条件
ANDNOT 12.08  ; 右机械手伸缩气缸
@LD W4.08  ; 伸缩气缸-HMI
AND T0016  ; 右机械手升降气缸缩回位时间
AND 12.08  ; 右机械手伸缩气缸
KEEP(011) W24.11  ; 右机械手伸缩气缸手动伸出
; rung 14
@LD W4.07  ; 升降气缸-HMI
AND 24.04  ; 右机械手伸缩气缸伸出条件
AND T0019  ; 右机械手伸缩气缸伸出位时间
ANDNOT 12.07  ; 右机械手升降气缸
@LD W4.07  ; 升降气缸-HMI
AND 12.07  ; 右机械手升降气缸
KEEP(011) W24.12  ; 右机械手升降气缸手动伸出

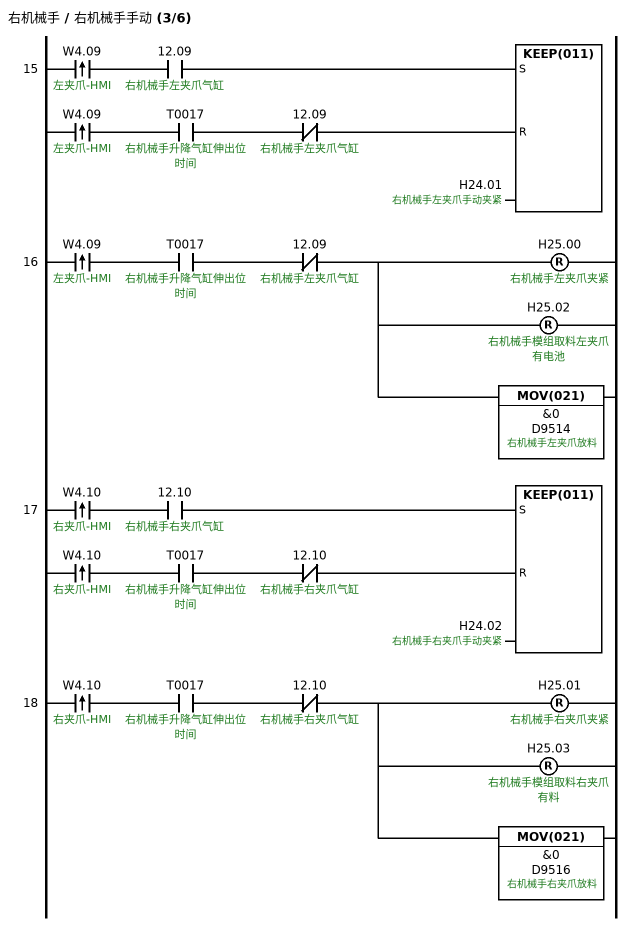
; rung 15
@LD W4.09  ; 左夹爪-HMI
AND 12.09  ; 右机械手左夹爪气缸
@LD W4.09  ; 左夹爪-HMI
AND T0017  ; 右机械手升降气缸伸出位时间
ANDNOT 12.09  ; 右机械手左夹爪气缸
KEEP(011) H24.01  ; 右机械手左夹爪手动夹紧
; rung 16
@LD W4.09  ; 左夹爪-HMI
AND T0017  ; 右机械手升降气缸伸出位时间
ANDNOT 12.09  ; 右机械手左夹爪气缸
RSET H25.00  ; 右机械手左夹爪夹紧
RSET H25.02  ; 右机械手模组取料左夹爪有电池
MOV(021) &0 D9514  ; 右机械手左夹爪放料
; rung 17
@LD W4.10  ; 右夹爪-HMI
AND 12.10  ; 右机械手右夹爪气缸
@LD W4.10  ; 右夹爪-HMI
AND T0017  ; 右机械手升降气缸伸出位时间
ANDNOT 12.10  ; 右机械手右夹爪气缸
KEEP(011) H24.02  ; 右机械手右夹爪手动夹紧
; rung 18
@LD W4.10  ; 右夹爪-HMI
AND T0017  ; 右机械手升降气缸伸出位时间
ANDNOT 12.10  ; 右机械手右夹爪气缸
RSET H25.01  ; 右机械手右夹爪夹紧
RSET H25.03  ; 右机械手模组取料右夹爪有料
MOV(021) &0 D9516  ; 右机械手右夹爪放料

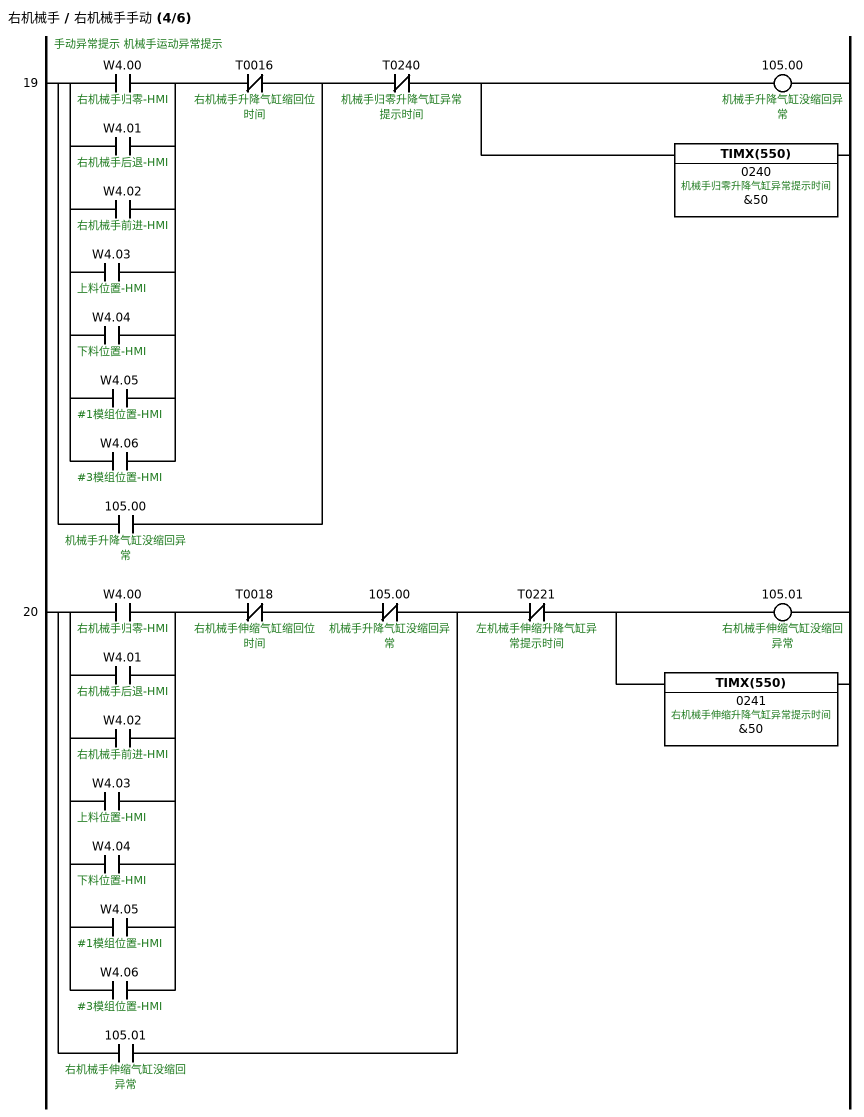
; rung 19: 手动异常提示 机械手运动异常提示
LD W4.00  ; 右机械手归零-HMI
OR W4.01  ; 右机械手后退-HMI
OR W4.02  ; 右机械手前进-HMI
OR W4.03  ; 上料位置-HMI
OR W4.04  ; 下料位置-HMI
OR W4.05  ; #1模组位置-HMI
OR W4.06  ; #3模组位置-HMI
ANDNOT T0016  ; 右机械手升降气缸缩回位时间
OR 105.00  ; 机械手升降气缸没缩回异常
ANDNOT T0240  ; 机械手归零升降气缸异常提示时间
OUT 105.00  ; 机械手升降气缸没缩回异常
TIMX(550) 0240 &50  ; 机械手归零升降气缸异常提示时间
; rung 20
LD W4.00  ; 右机械手归零-HMI
OR W4.01  ; 右机械手后退-HMI
OR W4.02  ; 右机械手前进-HMI
OR W4.03  ; 上料位置-HMI
OR W4.04  ; 下料位置-HMI
OR W4.05  ; #1模组位置-HMI
OR W4.06  ; #3模组位置-HMI
ANDNOT T0018  ; 右机械手伸缩气缸缩回位时间
ANDNOT 105.00  ; 机械手升降气缸没缩回异常
OR 105.01  ; 右机械手伸缩气缸没缩回异常
ANDNOT T0221  ; 左机械手伸缩升降气缸异常提示时间
OUT 105.01  ; 右机械手伸缩气缸没缩回异常
TIMX(550) 0241 &50  ; 右机械手伸缩升降气缸异常提示时间

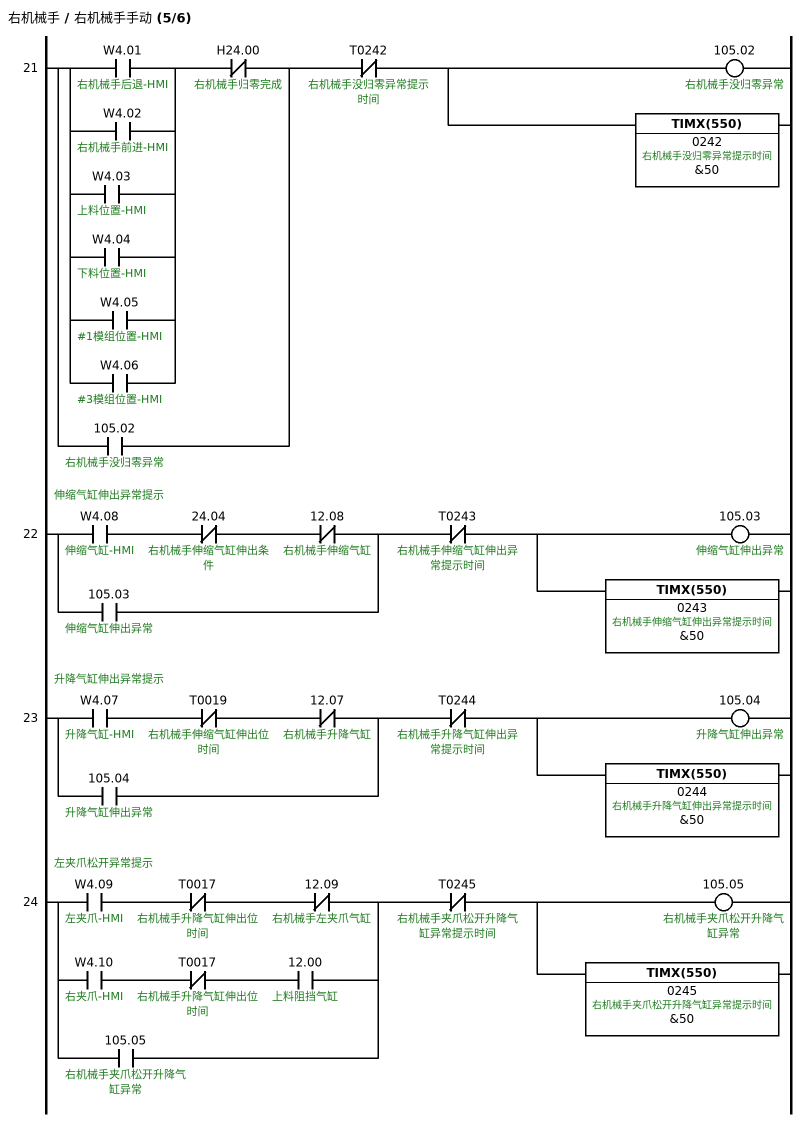
; rung 21
LD W4.01  ; 右机械手后退-HMI
OR W4.02  ; 右机械手前进-HMI
OR W4.03  ; 上料位置-HMI
OR W4.04  ; 下料位置-HMI
OR W4.05  ; #1模组位置-HMI
OR W4.06  ; #3模组位置-HMI
ANDNOT H24.00  ; 右机械手归零完成
OR 105.02  ; 右机械手没归零异常
ANDNOT T0242  ; 右机械手没归零异常提示时间
OUT 105.02  ; 右机械手没归零异常
TIMX(550) 0242 &50  ; 右机械手没归零异常提示时间
; rung 22: 伸缩气缸伸出异常提示
LD W4.08  ; 伸缩气缸-HMI
ANDNOT 24.04  ; 右机械手伸缩气缸伸出条件
ANDNOT 12.08  ; 右机械手伸缩气缸
OR 105.03  ; 伸缩气缸伸出异常
ANDNOT T0243  ; 右机械手伸缩气缸伸出异常提示时间
OUT 105.03  ; 伸缩气缸伸出异常
TIMX(550) 0243 &50  ; 右机械手伸缩气缸伸出异常提示时间
; rung 23: 升降气缸伸出异常提示
LD W4.07  ; 升降气缸-HMI
ANDNOT T0019  ; 右机械手伸缩气缸伸出位时间
ANDNOT 12.07  ; 右机械手升降气缸
OR 105.04  ; 升降气缸伸出异常
ANDNOT T0244  ; 右机械手升降气缸伸出异常提示时间
OUT 105.04  ; 升降气缸伸出异常
TIMX(550) 0244 &50  ; 右机械手升降气缸伸出异常提示时间
; rung 24: 左夹爪松开异常提示
LD W4.09  ; 左夹爪-HMI
ANDNOT T0017  ; 右机械手升降气缸伸出位时间
ANDNOT 12.09  ; 右机械手左夹爪气缸
LD W4.10  ; 右夹爪-HMI
ANDNOT T0017  ; 右机械手升降气缸伸出位时间
AND 12.00  ; 上料阻挡气缸
ORLD
OR 105.05  ; 右机械手夹爪松开升降气缸异常
ANDNOT T0245  ; 右机械手夹爪松开升降气缸异常提示时间
OUT 105.05  ; 右机械手夹爪松开升降气缸异常
TIMX(550) 0245 &50  ; 右机械手夹爪松开升降气缸异常提示时间

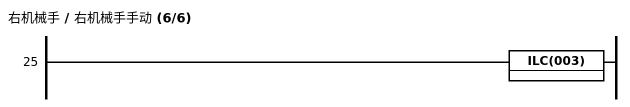
; rung 25
ILC(003)

### Section 右机械手自动

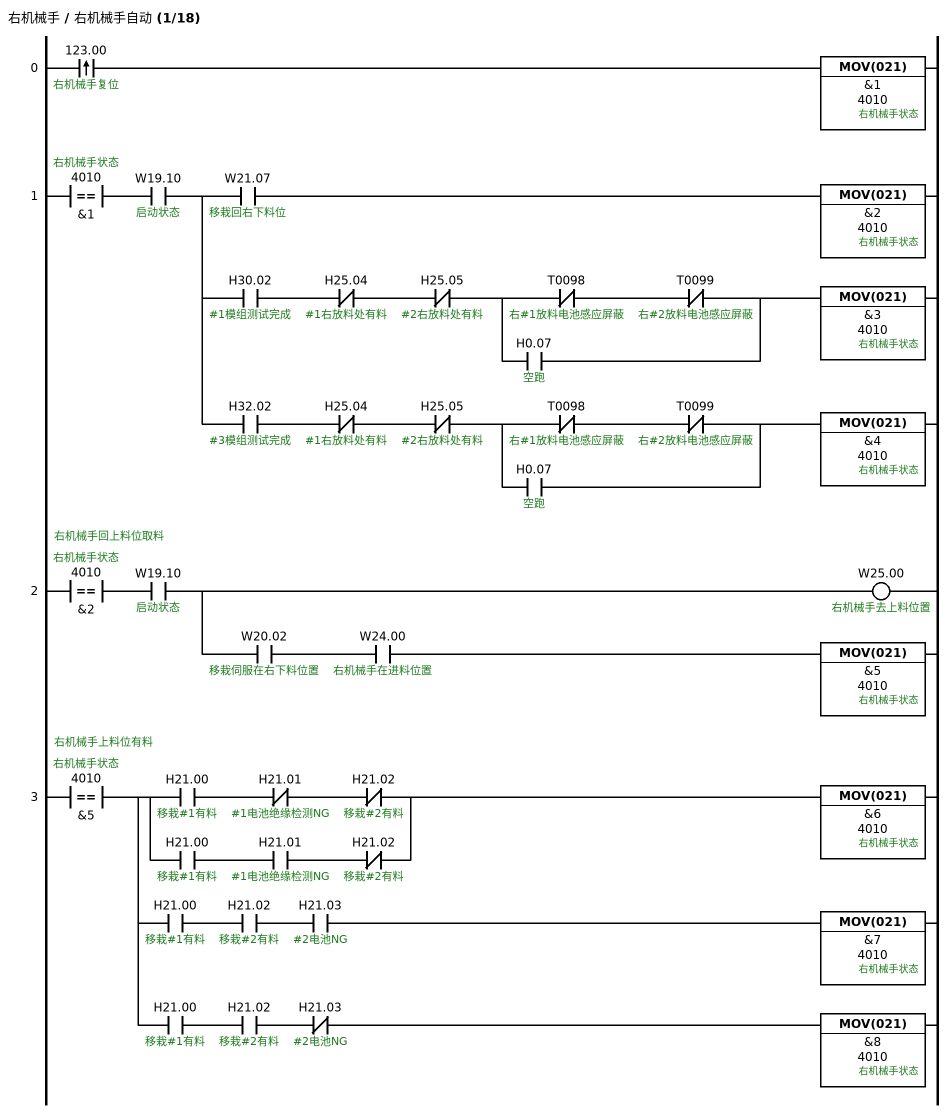
; rung 0
@LD 123.00  ; 右机械手复位
MOV(021) &1 4010  ; 右机械手状态
; rung 1
LD=(300) 4010 &1  ; 右机械手状态
AND W19.10  ; 启动状态
OUT TR0
AND W21.07  ; 移栽回右下料位
MOV(021) &2 4010  ; 右机械手状态
LD TR0
AND H30.02  ; #1模组测试完成
ANDNOT H25.04  ; #1右放料处有料
ANDNOT H25.05  ; #2右放料处有料
LDNOT T0098  ; 右#1放料电池感应屏蔽
ANDNOT T0099  ; 右#2放料电池感应屏蔽
OR H0.07  ; 空跑
ANDLD
MOV(021) &3 4010  ; 右机械手状态
LD TR0
AND H32.02  ; #3模组测试完成
ANDNOT H25.04  ; #1右放料处有料
ANDNOT H25.05  ; #2右放料处有料
LDNOT T0098  ; 右#1放料电池感应屏蔽
ANDNOT T0099  ; 右#2放料电池感应屏蔽
OR H0.07  ; 空跑
ANDLD
MOV(021) &4 4010  ; 右机械手状态
; rung 2: 右机械手回上料位取料
LD=(300) 4010 &2  ; 右机械手状态
AND W19.10  ; 启动状态
OUT W25.00  ; 右机械手去上料位置
AND W20.02  ; 移栽伺服在右下料位置
AND W24.00  ; 右机械手在进料位置
MOV(021) &5 4010  ; 右机械手状态
; rung 3: 右机械手上料位有料
LD=(300) 4010 &5  ; 右机械手状态
OUT TR0
LD H21.00  ; 移栽#1有料
ANDNOT H21.01  ; #1电池绝缘检测NG
ANDNOT H21.02  ; 移栽#2有料
LD H21.00  ; 移栽#1有料
AND H21.01  ; #1电池绝缘检测NG
ANDNOT H21.02  ; 移栽#2有料
ORLD
ANDLD
MOV(021) &6 4010  ; 右机械手状态
LD TR0
AND H21.00  ; 移栽#1有料
AND H21.02  ; 移栽#2有料
AND H21.03  ; #2电池NG
MOV(021) &7 4010  ; 右机械手状态
LD TR0
AND H21.00  ; 移栽#1有料
AND H21.02  ; 移栽#2有料
ANDNOT H21.03  ; #2电池NG
MOV(021) &8 4010  ; 右机械手状态

